PROGRAM MAIN
VAR
	stFRConnection : ST_FRConnection;
	fbFRPower : FB_FRPower;
	fbFRProgSelect : FB_FRProgSelect;
	
	bIMSTP : BOOL;
	bHold : BOOL;
	bSFSPD : BOOL;
	bCycleStop : BOOL;
	bFaultReset : BOOL;
	bStart : BOOL;
	bHome : BOOL;
	bEnable : BOOL;

	bCmdEnabled : BOOL;
	bSystemReady : BOOL;
	bPrgRunning : BOOL;
	bPrgPaused : BOOL;
	bMotionHeld : BOOL;
	bFault : BOOL;
	bAtPerch : BOOL;
	bTPEnabled : BOOL;
	bBattAlarm : BOOL;
	bBusy : BOOL;
	
	bProgSelectExec : BOOL;
	bProgSelectDone : BOOL;
	bProgSelectBusy : BOOL;
	nProgSelectNo : USINT;
	nSelectedProgNo : USINT;
END_VAR

FRTest();

ACTION FRTest:
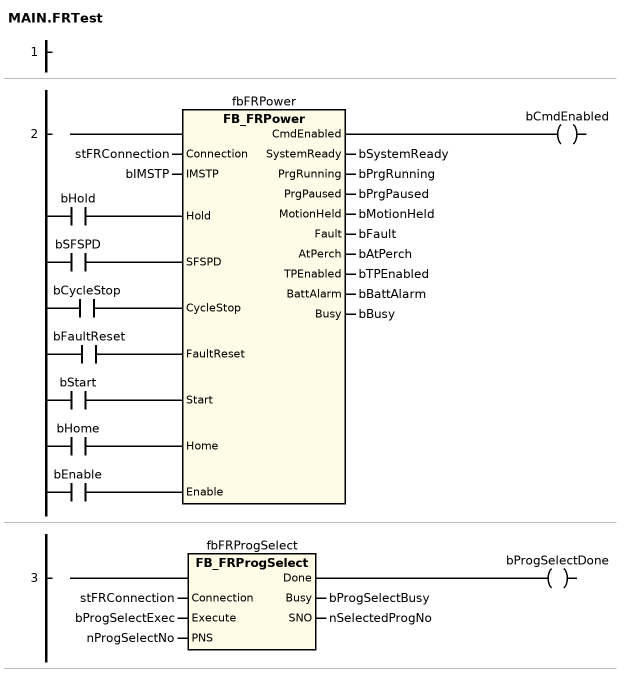
// NETWORK 1

// NETWORK 2
fbFRPower(
    Connection := stFRConnection,
    IMSTP := bIMSTP,
    Hold := bHold,
    SFSPD := bSFSPD,
    CycleStop := bCycleStop,
    FaultReset := bFaultReset,
    Start := bStart,
    Home := bHome,
    Enable := bEnable,
    SystemReady => bSystemReady,
    PrgRunning => bPrgRunning,
    PrgPaused => bPrgPaused,
    MotionHeld => bMotionHeld,
    Fault => bFault,
    AtPerch => bAtPerch,
    TPEnabled => bTPEnabled,
    BattAlarm => bBattAlarm,
    Busy => bBusy); // FB_FRPower
bCmdEnabled := fbFRPower.CmdEnabled;

// NETWORK 3
fbFRProgSelect(
    Connection := stFRConnection,
    Execute := bProgSelectExec,
    PNS := nProgSelectNo,
    Busy => bProgSelectBusy,
    SNO => nSelectedProgNo); // FB_FRProgSelect
bProgSelectDone := fbFRProgSelect.Done;
END_ACTION

END_PROGRAM

(* stored: Version 1.1.0.1, ProductVersion 3.1.4024.15
   POU MAIN: Id {e81fdd85-a5af-4a5b-903d-7a3802be9cd8}, SpecialFunc None
   Action FRTest: Id {cd9a0e6c-7701-4984-9c62-bc81f0bd8728} *)
